Staubli VAL3: getView.pgx

public program getView(bool& x_bView[])
begin
  //-----------------------------------------------------------------------
  //Header begin
  //Description of program
  //  This program returns true in x_bView if the menu of the list
  //  is displayed in full-page and false otherwise.
  //  这个程序当整个菜单列表全屏显示的时候，返回在x_bView的真值，否则为假。
  //Output parameters  输出参数
  //  bool x_bView : 布尔量x_bView
  //    role : Status of the size of list menu.
  //    作用：菜单列表的大小状态
  //    possible values : true when the list menu is displayed in full-page,
  //                      false otherwise.
  //    可能的值：当菜单列表全屏显示时，返回真值，否则为假。
  //Example
  //  call getView(l_bView)
  //
  //History
  //  Creation : 28-04-08 - f.Rob
  //Header end
  //-----------------------------------------------------------------------
  if nBottomX==38
    x_bView=true
  else
    x_bView=false
  endIf
end
